// TwinCAT 3 PLC project TC_Sample
// ProgramVersion: 3.1.0.5
// libraries:
//   Tc2_Standard, * (Beckhoff Automation GmbH)
//   Tc2_System, * (Beckhoff Automation GmbH)
//   Tc2_Utilities, * (Beckhoff Automation GmbH)
//   Tc3_JsonXml, * (Beckhoff Automation GmbH)
//   Tc3_Module, * (Beckhoff Automation GmbH)
//   Util, * (System)
//   Tc2_ControllerToolbox,newest,Beckhoff Automation GmbH
//   Tc2_TempController,newest,Beckhoff Automation GmbH
//   VisuSymbols,3.5.10.0,System
// project tree:
//   DUTs/ E_Mode.TcTLEO, E_SelectedParameterSet.TcDUT, E_State.TcDUT, ST_AutoTuneGains.TcDUT
//   DUTs/HMI/ E_CTRL_MODE_HMI.TcDUT, E_CTRL_STATE_HMI.TcDUT
//   / GlobalTextList.TcGTLO, PlcTask.TcTTO, Visualization Manager.TcVMO (not stored)
//   POUs/Controller/ MAIN.TcPOU
//   POUs/ FB_Process.TcPOU
//   VISUs/ TL_Mode.TcTLO, TL_SelectedParameterSet.TcTLO, Visualization.TcVIS
// real-time tasks:
//   TASK PlcTask: cycle T#10ms, priority 20, ADS port 350

CONFIGURATION TC_Sample
    RESOURCE PLC ON TwinCAT3
        TASK PlcTask(INTERVAL := T#1ms, PRIORITY := 20);
        PROGRAM MAIN WITH PlcTask : MAIN;
    END_RESOURCE
END_CONFIGURATION

// ---- DUTs/E_Mode.TcTLEO
{attribute 'qualified_only'}
{attribute 'strict'}
{attribute 'to_string'}
TYPE E_Mode :
(
	Tune 	:=0,
	Run		:=1
);
END_TYPE

// ---- DUTs/E_SelectedParameterSet.TcDUT
{attribute 'qualified_only'}
{attribute 'strict'}
{attribute 'to_string'}
TYPE E_SelectedParameterSet :
(
	Fast := 0,
	Slow :=1,
	Asymptotic :=2
);
END_TYPE

// ---- DUTs/E_State.TcDUT
{attribute 'qualified_only'}
{attribute 'strict'}
{attribute 'to_string'}
TYPE E_State :
(
	Idel:=0		,
	LoadTunningParmaeters:=1,
	AutoTuneInProgress:=2,
	LoadRunParameters:=3,
	Run:=4,
	Error:=5,
	Reset:=6
);
END_TYPE

// ---- DUTs/HMI/E_CTRL_MODE_HMI.TcDUT
{attribute 'qualified_only'}
{attribute 'to_string'}
TYPE E_CTRL_MODE_HMI :
(
	IDLE:=0,
	PASSIVE, 
	ACTIVE, 
	RESET, 
	MANUAL, 
	TUNE, 
	SELFTEST,  
	SYNC_MOVEMENT,
	FREEZE 
);
END_TYPE

// ---- DUTs/HMI/E_CTRL_STATE_HMI.TcDUT
{attribute 'qualified_only'}
{attribute 'to_string'}
TYPE E_CTRL_STATE_HMI :
(
	IDLE,  
	PASSIVE, 
	ACTIVE,
	RESET,
	MANUAL,
	TUNING,
	TUNED,
	SELFTEST,
	ERROR, 
	SYNC_MOVEMENT,
	FREEZE 
);
END_TYPE

// ---- DUTs/ST_AutoTuneGains.TcDUT
TYPE ST_AutoTuneGains :
STRUCT
	fKp					:LREAL;
	fTn					:LREAL;
	fTv					:LREAL;
	fTd					:LREAL;	
END_STRUCT
END_TYPE

// ---- POUs/Controller/MAIN.TcPOU
PROGRAM MAIN
VAR
		(* Controller *)
		eCTRL_ModeController 	: E_CTRL_MODE := E_CTRL_MODE.eCTRL_MODE_IDLE;
		
		fW						: LREAL	:= 100.0;				(* setpoint *)
		fY						: LREAL;						(* control value *)
		fX						: LREAL;						(* actual value from simulated process *)
		
	
		stControllerParameter	: ST_CTRL_TempCtrlParameter := (		
		
			(* general parameters 													 *)
			iMode					:= 1,											(* 1=heating, 2=cooling, 3=heating&cooling *)
			iReactionOnFailure		:= eCTRL_ReactionOnFailure_StopController,		(* 0=controller off, 1=manual op, 2=yMin, 3=yMax *)
	    	
			bSelCtrlParameterSet	:= FALSE,										(* FALSE = internal set, TRUE = external set *)//Internal are calculated after an auto tune
	    	
			dwAlarmSupp				:= 16#0000EFFF,									(* alarm suppression *)
			tCtrlCycleTime			:= T#10MS,										(* controller cycle time *)
			tTaskCycleTime			:= T#10MS,										(* plc task cycle time *)
			
			(* tuning parameters 													 *)
			iTuningMode				:= 1,											(* only heating, only cooling, first heating then cooling or vice versa *)
	    	
			tTuneStabilisation		:= T#5S,										(* wait for a stable system *)
	    	
			fEndTunePercentHeating	:= 80.0,										(* switch to closed loop control when X > 0.8*W *)
			fYTuneHeating			:= 100.0,										(* step change while tuning operation *)
			fYStableHeating			:= 0.0,											(* tuning operation *)
	    	
			fEndTunePercentCooling	:= 20.0,										(* switch to closed loop control when X < 0.2*W *)
			fYTuneCooling			:= 0.0,											(* step change while tuning operation *)
			fYStableCooling			:= 0.0,											(* tuning operation *)
			fScalingFactor			:= 1.0,											(* Scaling factor for KP heating/cooling *)
			
			(* setpoint parameters 													 *)
			fWMin					:= 0.0,											(* lower limit *)
			fWMax					:= 300.0,										(* upper limit *)
	    	
			(* start up *)
			bEnableSoftStart		:= FALSE,										(* FALSE = no soft start, TRUE = soft start *)
			bEnableRamping			:= FALSE,										(* FALSE = no ramping, TRUE = ramping *)
	    	
			fWStartUp				:= 0.0,											(* soft start plateau setpoint *)
			tStartUp				:= T#0MS,										(* soft start waiting time*)
			bStartUpRamping			:= FALSE,										(* enable ramping while start up phase *)
			fWStartUpVeloPos		:= 1.0,											(* max gradient for increasing setpoint in start up phase*)
			fWStartUpVeloNeg		:= 1.0,											(* max gradient for decreasing setpoint in start up phase *)
	    	
			fWVeloPos				:= 1.0,											(* max gradient for increasing setpoint *)
			fWVeloNeg				:= 1.0,											(* max gradient for decreasing setpoint *)	
	    	
			(* actual value parameters     											 *)
			bFilter 				:= FALSE,
			tFilter					:= T#0S,
			
			(* deadband parameters     												 *)
			bDeadband				:= FALSE,
			fEDeadband				:= 0.0,											(* deadband *)
			
			(* control value parameters     										 *)
			fYMin					:= 0.0,											(* lower limit *)
			fYMax					:= 100.0,										(* upper limit *)
			fYManual				:= 0.0,									 		(* manual operation*)
			fYOnFailure				:= 0.0,											(* control value on failure *)
	    	
			tPWMCycleTime			:= t#1s,										(* PWM: period *)
			tPWMMinOffTime			:= t#0s,										(* PWM: min off time *)
			tPWMMinOnTime			:= t#0s,										(* PWM: min on time *)
			tPWMWaitingTime			:= t#0s,										(* PWM: min waiting time *) (* not yet implemented !!!!*)
	    	
			fYThresholdOff			:= 0.0,											(* 3-Point: Off threshold *)
			fYThresholdOn			:= 0.0,											(* 3-Point: On threshold *)
	    	
			nCyclesForSwitchOver	:= 100,
	    	
			(* controller settings			     									 *)
			bEnablePreController 	:= FALSE,										(* enable precontroller *)
			bEnableZones 			:= FALSE,										(* enable zone around setpoint with open loop control *)
			bEnableCVFilter 		:= FALSE,										(* enable filter for CV (type see iFilterType) *)
			iFilterType 			:= E_CTRL_FilterType.eCTRL_FilterType_FIRSTORDER,(* filtertype of CV filter *)
			iControllerType 		:= eCTRL_ControllerType_PID,					(* used controller normally PID *)
			
			
			(* min max temperatures	     											 *)
			TempLow					:= -5.0,
			TempLowLow				:= -10.0,
			TempHigh				:= 5.0,
			TempHighHigh			:= 10.0,
			TempAbsoluteHigh		:= 300.0,
			TempAbsoluteLow			:= 0.0,	
			
			(* internal tuning parameters *)
			fTuneKp					:= 1.2,
			fTuneTn					:= 2.0,
			fTuneTv					:= 0.42,
			fTuneTd					:= 0.25
		);
	
		
	fbTempController			: FB_CTRL_TempController;
	

	stController				: ST_CTRL_ParaController;
	
	Start					:BOOL;
	rtStart					:R_TRIG;
	Stop					:BOOL;
	rtStop					:R_TRIG;
	Reset					:BOOL;
	rtReset					:R_TRIG;
	State					:E_State;
	sState					:STRING;
	Mode					:E_Mode;
	SelectedParameterSet	:E_SelectedParameterSet;
	
	(* Simulate process *)	
	ResetProcess			:BOOL;
	ResetProcessStep		:INT;
	rtResetProcess			:R_TRIG;
	eCTRL_ModeProcess	 	: E_CTRL_MODE := E_CTRL_MODE.eCTRL_MODE_ACTIVE; 	
	fbProcess				: FB_Process;		
	
	
	(*HMI*)
	eControllerModeHMI			:E_CTRL_MODE_HMI;
	sControllerMode				:STRING;
	eControllerState			:E_CTRL_STATE_HMI;
	sControllerState			:STRING;
	
	eProcessModeHMI				:E_CTRL_MODE_HMI;
	sProcessModeHMI				:STRING;
	eProcessStateHMI			:E_CTRL_STATE_HMI;
	sProcessStateHMI			:STRING;
	
	////Test case
	//bStartTest				: BOOL;
	//iTestSetp				: UDINT;
	//tonReset				: TON;
	//tonRun					: TON;	
	//stTestResults			: ST_TestResults;
	
	//Write results to a file
	//fbJsonFile				:FB_AppendJsonObjectToArrayAndWriteToFile;
   	//sFilePath      			:T_MaxString := 'C:\TwinCAT\3.1\Boot\TestResults.json';
	//
	//Recipe manager
	//sRecipeLoaded			:STRING;
	//RecipeMan				:RecipeManCommands;
	//{attribute 'displaymode':='hex'}
	//ResultOfLoad			:DWORD;
	//iRecipeIndex			:UDINT;
END_VAR
VAR PERSISTENT
	arControllerParams		:ARRAY[E_SelectedParameterSet.Fast..E_SelectedParameterSet.Asymptotic] OF ST_CTRL_ParaController; 
END_VAR
VAR CONSTANT
	arAutoTuneGains			: ARRAY [E_SelectedParameterSet.Fast..E_SelectedParameterSet.Asymptotic] OF ST_AutoTuneGains := [(fKp := 1.2, fTn := 2, fTv := 0.42, fTd := 0.25), (fKp := 1, fTn := 2.5, fTv := 0.42, fTd := 0.25), (fKp := 0.5, fTn := 3, fTv := 1, fTd := 0.25)];
END_VAR

(* Simulate process *)
rtResetProcess(CLK:=ResetProcess);
CASE ResetProcessStep OF
	0:
		IF rtResetProcess.Q THEN
			eCTRL_ModeProcess					:=E_CTRL_MODE.eCTRL_MODE_RESET;
			ResetProcessStep:=10;
		END_IF
		
	10:
		IF fbProcess.eState = E_CTRL_STATE.eCTRL_STATE_IDLE THEN
			eCTRL_ModeProcess					:=E_CTRL_MODE.eCTRL_MODE_ACTIVE;
			ResetProcessStep:=0;
		END_IF
END_CASE

fbProcess(	eCTRL_Mode	:= eCTRL_ModeProcess,
			fY 			:= fbTempController.fYAnalog, 
			bNoise 		:= , 
			tTa 		:= stControllerParameter.tTaskCycleTime);	
			
			
			

(* Actual temperature *)				
fX := fbProcess.fX;	

(* Controller *)
fbTempController(
					eCtrlMode				:= eCTRL_ModeController, 
					bSelSetpoint			:= FALSE, 
					fW1						:= fW, 
					fW2						:= , 
					fX						:= fX, 
					fYManual				:= , 
					bOpenThermocouple		:= FALSE, 
					bReverseThermocouple	:= FALSE, 
					bBackVoltage			:= FALSE, 
					bLeakage				:= FALSE, 
					bShortCircuit			:= FALSE, 
					bOpenCircuit			:= FALSE, 
					sParaControllerExternal	:= stController, 
					sControllerParameter	:= stControllerParameter, 
					);
					 
(* Analog output *)			
fY 			:= fbTempController.fYAnalog;

rtStart(CLK:=Start);
rtStop(CLK:=Stop);
rtReset(CLK:=Reset);

CASE State OF 
	E_State.Idel:		
		IF rtStart.Q THEN
			CASE Mode OF 
				E_Mode.Tune:
					State:=E_State.LoadTunningParmaeters;
				E_Mode.Run:
					State:=E_State.LoadRunParameters;
			END_CASE
		ELSIF fbTempController.eCtrlState = E_CTRL_STATE.eCTRL_STATE_ERROR THEN
			State								:=E_State.Error;
		ELSIF rtReset.Q THEN
			State:=E_State.Reset;
		END_IF
		
	E_State.LoadTunningParmaeters:
			stControllerParameter.bSelCtrlParameterSet:=FALSE;
			
			stControllerParameter.fTuneKp:=arAutoTuneGains[SelectedParameterSet].fKp;
			stControllerParameter.fTuneTd:=arAutoTuneGains[SelectedParameterSet].fTd;
			stControllerParameter.fTuneTv:=arAutoTuneGains[SelectedParameterSet].fTv;
			stControllerParameter.fTuneTd:=arAutoTuneGains[SelectedParameterSet].fTd;
			
			eCTRL_ModeController				:=E_CTRL_MODE.eCTRL_MODE_TUNE;
			State								:=E_State.AutoTuneInProgress;
			
	E_State.AutoTuneInProgress:
	
		IF fbTempController.eCtrlState = E_CTRL_STATE.eCTRL_STATE_TUNED THEN		
			//Grab the calculated internal gains from the auto tune, and save them off to a persistent variable
			arControllerParams[SelectedParameterSet]:= fbTempController.sParaControllerInternal;
			eCTRL_ModeController 					:=E_CTRL_MODE.eCTRL_MODE_ACTIVE;
			State									:=E_State.Run;
		ELSIF fbTempController.eCtrlState = E_CTRL_STATE.eCTRL_STATE_ERROR THEN
			State									:=E_State.Error;
		END_IF
		
	E_State.LoadRunParameters:
		//Use "sParaControllerExternal"
		stControllerParameter.bSelCtrlParameterSet:=TRUE;
		stController:=arControllerParams[SelectedParameterSet];
		State									:=E_State.Run;
	
	E_State.Run:	
		eCTRL_ModeController 					:=E_CTRL_MODE.eCTRL_MODE_ACTIVE;
		
		IF fbTempController.eCtrlState = E_CTRL_STATE.eCTRL_STATE_ERROR THEN
			State								:=E_State.Error;
		END_IF
		
		IF rtStop.Q THEN
			eCTRL_ModeController				:=E_CTRL_MODE.eCTRL_MODE_IDLE;
			State								:=E_State.Idel;
		END_IF
		
	E_State.Error:
		IF rtReset.Q THEN
			State:=E_State.Reset;
		END_IF
		
	E_State.Reset:
		eCTRL_ModeController				:=E_CTRL_MODE.eCTRL_MODE_RESET;
		
		IF fbTempController.eCtrlState=E_CTRL_STATE.eCTRL_STATE_IDLE THEN
			eCTRL_ModeController				:=E_CTRL_MODE.eCTRL_MODE_IDLE;
			State								:=E_State.Idel;
		END_IF
END_CASE





(*HMI*)
eControllerModeHMI:=fbTempController.eCtrlMode;
sControllerMode:=TO_STRING(eControllerModeHMI);

eControllerState:=fbTempController.eCtrlState;
sControllerState:=TO_STRING(eControllerState);

eProcessModeHMI:=fbProcess.eCTRL_Mode;
sProcessModeHMI:=TO_STRING(eProcessModeHMI);

eProcessStateHMI:=fbProcess.eState;
sProcessStateHMI:=TO_STRING(eProcessStateHMI);

sState:=TO_STRING(State);

//Test case
//CASE iTestSetp OF
//	0://Idel
//		IF bStartTest THEN
//			iRecipeIndex:=0;
//			fbJsonFile.ResetDocument();
//			bStartTest	:=FALSE;
//			iTestSetp	:=5;
//		END_IF
//		
//	5: //Load recipe or finish
//		CASE iRecipeIndex OF
//			0:sRecipeLoaded:='Fast';
//			1:sRecipeLoaded:='Slow';
//			2:sRecipeLoaded:='Asymptotic';				
//		END_CASE
//			stTestResults.TestName:=sRecipeLoaded;
//			
//		CASE iRecipeIndex OF
//			0..2:	
//				ResultOfLoad:=RecipeMan.WriteRecipe(RecipeDefinitionName:='AutoTuneParms', RecipeName:=sRecipeLoaded);
//				IF ResultOfLoad = 0 THEN
//					MEMSET(ADR(stTestResults),0,SIZEOF(stTestResults));
//					stTestResults.InitialParmsUsed 		:=stControllerParameter;
//					iTestSetp							:=10;
//				ELSE
//					iTestSetp:=99;
//				END_IF
//			ELSE
//				iTestSetp:=100;
//		END_CASE
//		
//		
//	10://Waiting for controller to complete auto tuning	
//		eCTRL_ModeController				:=E_CTRL_MODE.eCTRL_MODE_TUNE;
//		eCTRL_ModeProcess					:=E_CTRL_MODE.eCTRL_MODE_ACTIVE;
//		
//		IF fbTempController.eCtrlState = E_CTRL_STATE.eCTRL_STATE_TUNED THEN	
//			eCTRL_ModeController 				:=E_CTRL_MODE.eCTRL_MODE_ACTIVE;
//			stTestResults.CalcedInternalGains	:= fbTempController.sParaControllerInternal;
//			iTestSetp							:=20;
//		END_IF
//		
//	20: //Finished auto tunning - run for a bit to see results of switching from auto tune to active	
//		tonRun(IN:=TRUE,PT := TIME#3M);
//		IF tonRun.Q THEN
//			stTestResults.MaxOverShootDuringAutoTune:= fbTempController.fMaxOverShoot;
//			stTestResults.StartupTimeDuringAutoTune := fbTempController.tStartUpTime;
//			tonRun(IN:=FALSE);
//			iTestSetp:=30;
//		END_IF
//		
//	30://Reset simulation model, and controller
//		eCTRL_ModeController	:=E_CTRL_MODE.eCTRL_MODE_RESET;
//		eCTRL_ModeProcess		:=E_CTRL_MODE.eCTRL_MODE_RESET;
//		tonReset(IN:=TRUE,PT := TIME#5S);
//		IF tonReset.Q THEN
//			tonReset(IN:=FALSE);
//			iTestSetp		:=40;
//		END_IF
//		
//	40://Run test with calcuated gains from auto tuning
//		eCTRL_ModeController	:=E_CTRL_MODE.eCTRL_MODE_ACTIVE;
//		eCTRL_ModeProcess		:=E_CTRL_MODE.eCTRL_MODE_ACTIVE;
//		tonRun(IN:=TRUE, PT:= TIME#3M);
//		IF tonRun.Q THEN
//			stTestResults.MaxOverShoot	:=fbTempController.fMaxOverShoot;
//			stTestResults.StartupTime 	:=fbTempController.tStartUpTime;
//			fbJsonFile.AddObject(nData:=SIZEOF(stTestResults) , pData:=ADR(stTestResults));
//			tonRun(IN:=FALSE);
//			iTestSetp:=50;
//		END_IF		
//		
//	50://Fisned running test
//		eCTRL_ModeController	:=E_CTRL_MODE.eCTRL_MODE_RESET;
//		eCTRL_ModeProcess		:=E_CTRL_MODE.eCTRL_MODE_RESET;
//		iTestSetp				:=0;
//
//	
//	99://Error
//		iTestSetp:=0;	
//		
//	100://Test finished - save results to a file	
//		IF fbJsonFile.SaveDocumentToFile(sFilePath:=sFilePath , bSaved=> ) THEN
//			iTestSetp				:=0;
//		END_IF
//	
//END_CASE
//
//
//
//

END_PROGRAM

// ---- POUs/FB_Process.TcPOU
FUNCTION_BLOCK FB_Process

VAR_INPUT
	eCTRL_Mode  : E_CTRL_MODE;
	fY			:	LREAL;
	tTa			:	TIME;
	bNoise		:	BOOL;
END_VAR

VAR_OUTPUT
	fX		:	LREAL;
	eState	:E_CTRL_STATE;
END_VAR

VAR
	(* Processparameters *)
	tT11		:	TIME	:= T#10S; //T#5S;
	tT12		:	TIME	:= T#35S; //t#25s;

	(* process *)
	fbProcessPart1	:	FB_CTRL_PT1;
	fbProcessPart2	:	FB_CTRL_PT1;
	fbNoise			:	FB_CTRL_NOISE_GENERATOR;

	stProcessPart1	:	ST_CTRL_PT1_PARAMS;
	stProcessPart2	:	ST_CTRL_PT1_PARAMS;
	stNoise			:	ST_CTRL_NOISE_GENERATOR_PARAMS;
	
END_VAR

(* init structures *)
stProcessPart1.fKp :=1.2; //1.0;
stProcessPart1.tCtrlCycleTime := tTa;
stProcessPart1.tT1 := tT11;
stProcessPart1.tTaskCycleTime := tTa;

stProcessPart2.fKp := 1.2;//1.0;
stProcessPart2.tCtrlCycleTime := tTa;
stProcessPart2.tT1 := tT12;
stProcessPart2.tTaskCycleTime := tTa;

stNoise.fAmplitude := 1.0;
stNoise.tCtrlCycleTime := tTa;
stNoise.tTaskCycleTime := tTa;

(* calculate and simulate process *)

fbProcessPart1(
				fIn:= fY,
				fManSyncValue:= 0.0,
				bSync:= FALSE,
				eMode:=eCTRL_Mode,
				bHold:= FALSE,
				stParams:= stProcessPart1);

fbProcessPart2(
				fIn:= fbProcessPart1.fOut,
				fManSyncValue:= 0.0,
				bSync:= FALSE,
				eMode:= eCTRL_Mode,
				bHold:= FALSE,
				stParams:= stProcessPart2);

fbNoise(
		fManSyncValue:= 0.0,
		eMode:= eCTRL_Mode,
		stParams:= stNoise);

IF bNoise THEN
	fX := fbProcessPart2.fOut + 0.01*fbNoise.fOut;
ELSE
	fX := fbProcessPart2.fOut;
END_IF;

eState:=fbProcessPart2.eState;

END_FUNCTION_BLOCK

// ---- GlobalTextList.TcGTLO
TEXTLIST GlobalTextList
  13 = '%s'
  644 = 'Controller'
  776 = 'KpCool'
  985 = 'KpHeat'
  55 = 'Machine'
  307 = 'Mode'
  609 = 'Noise'
  713 = 'Parameter Set'
  225 = 'Process'
  193 = 'Reset'
  822 = 'Start'
  187 = 'Start Auto Tune'
  127 = 'State'
  986 = 'Stop'
  343 = 'TdCool'
  116 = 'TdHeat'
  568 = 'TnCool'
  369 = 'TnHeat'
  727 = 'TvCool'
  485 = 'TvHeat'
END_TEXTLIST

// ---- VISUs/TL_Mode.TcTLO
TEXTLIST TL_Mode
  0 = 'Tune'
  1 = 'Run'
   = ''
END_TEXTLIST

// ---- VISUs/TL_SelectedParameterSet.TcTLO
TEXTLIST TL_SelectedParameterSet
  0 = 'Fast'
  1 = 'Slow'
  2 = 'Asymptotic'
   = ''
END_TEXTLIST

// ---- VISUs/Visualization.TcVIS
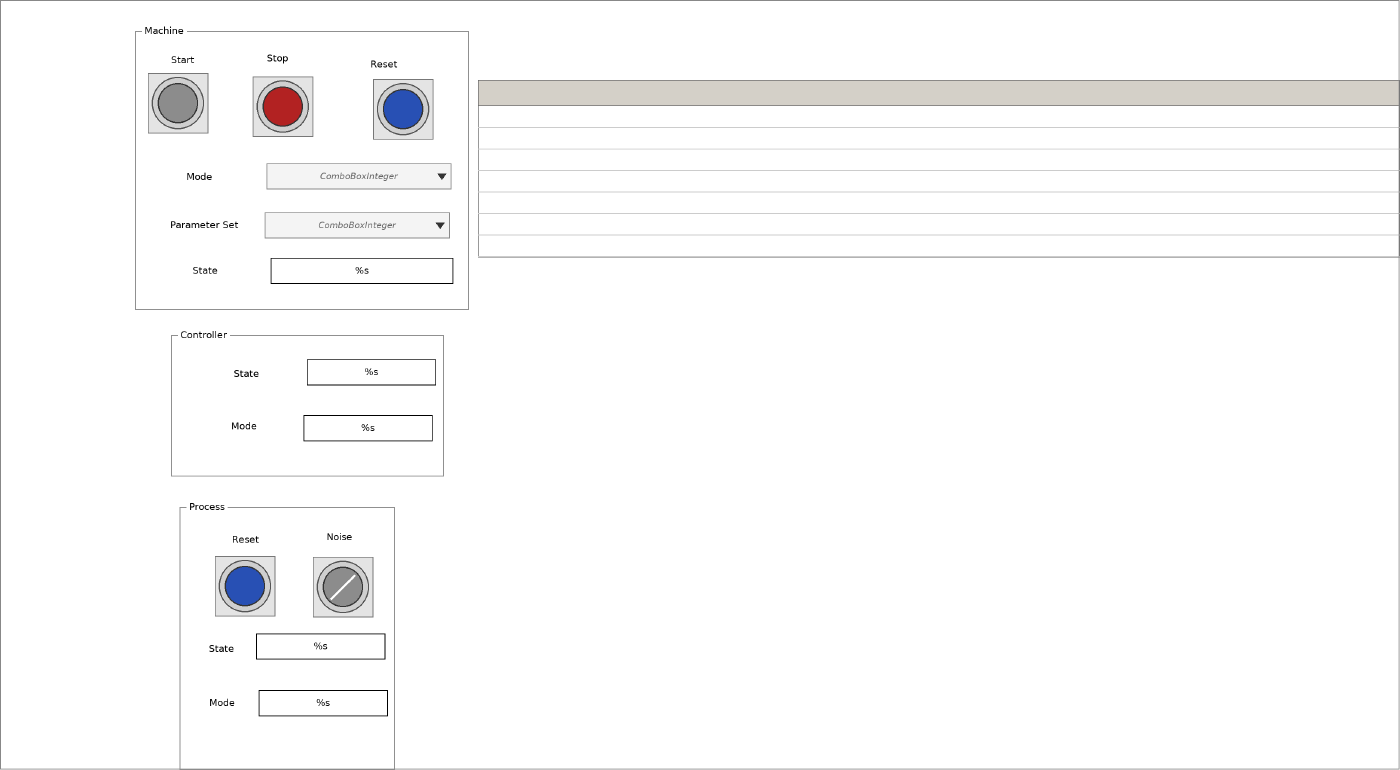
VISUALIZATION Visualization  // 1629x896
    GroupBox (199,382 317x172), "Controller"
        Rectangle (158,36 150x30), "%s", text variable: MAIN.sControllerState
        Label (13,38 150x30), "State"
        Label (10,99 150x30), "Mode"
        Rectangle (154,101 150x30), "%s", text variable: MAIN.sControllerMode
    GroupBox (209,582 250x314), "Process"
        PushSwitch (41,65 70x70), variable: MAIN.ResetProcess, behaviour: TAP, style: Switch-PushSwitch-Blue
        RotarySwitch (155,66 70x70), variable: MAIN.fbProcess.bNoise, behaviour: TOGGLE, style: Switch-RotarySwitch-Gray
        Label (2,31 150x30), "Reset"
        Rectangle (89,155 150x30), "%s", text variable: MAIN.sProcessStateHMI
        Rectangle (92,221 150x30), "%s", text variable: MAIN.sProcessModeHMI
        Label (145,28 82x30), "Noise"
        Label (13,158 72x30), "State"
        Label (9,221 81x30), "Mode"
    GroupBox (157,28 388x332), "Machine"
        PushSwitch (15,57 70x70), variable: MAIN.Start, behaviour: TAP, style: Switch-PushSwitch-Gray
        PushSwitch (137,61 70x70), variable: MAIN.Stop, behaviour: TAP, style: Switch-PushSwitch-Red
        Label (91,25 150x30), "Stop"
        PushSwitch (277,64 70x70), variable: MAIN.Reset, behaviour: TAP, style: Switch-PushSwitch-Blue
        Label (215,32 150x30), "Reset"
        ComboBoxInteger (153,162 215x30), variable: MAIN.Mode, text list: 'TL_Mode'
        Label (0,163 150x30), "Mode"
        ComboBoxInteger (151,219 215x30), variable: MAIN.SelectedParameterSet, text list: 'TL_SelectedParameterSet'
        Rectangle (158,272 212x30), "%s", text variable: MAIN.sState
        Label (7,272 150x30), "State"
        Label (10,27 91x30), "Start"
        Label (6,219 150x30), "Parameter Set"
    Table (556,93 1073x206), data array: MAIN.arControllerParams
        p3854506369: MAIN.arControllerParams[INDEX].KpHeat
        p1892666644: MAIN.arControllerParams[INDEX].TnHeat
        p338671338: MAIN.arControllerParams[INDEX].TvHeat
        p2170511999: MAIN.arControllerParams[INDEX].TdHeat
        p3723444502: MAIN.arControllerParams[INDEX].KpCool
        p1218418051: MAIN.arControllerParams[INDEX].TnCool
        p746581629: MAIN.arControllerParams[INDEX].TvCool
        p3104783080: MAIN.arControllerParams[INDEX].TdCool
END_VISUALIZATION
